// SIMATIC S7-200 project (STEP 7-Micro/WIN), CPU 224 CN REL 02.01

ORGANIZATION_BLOCK MAIN:OB1
TITLE=程序注释
BEGIN
Network 1 // 网络标题
// 网络注释
LD     SM0.1
R      M3.0, 8
R      Q0.0, 10
Network 2
LD     M1.0
R      M1.1, 1
Network 3
LD     M1.1
EU
R      M1.0, 1
R      M3.0, 8
R      Q0.0, 10
Network 4
LD     M1.1
ED
LD     M1.0
EU
OLD
R      M4.5, 2
R      Q0.5, 2
Network 5
LD     M1.1
CALL   SBR_0:SBR0
JMP    15
Network 6
LD     M1.0
EU
A      I0.4
R      M3.0, 8
R      Q0.0, 16
Network 7
LD     M1.0
EU
S      Q0.0, 1
Network 8
LD     M0.0
ED
R      M3.0, 8
R      Q0.0, 16
R      T33, 8
Network 9
LD     M0.0
A      M1.0
AN     M3.4
AN     M3.5
AN     M3.6
AN     M3.7
TON    T37, VW104
Network 10
LD     I0.0
LD     T37
A      M0.0
OLD
R      Q0.0, 1
A      M1.0
AN     Q0.5
AN     M3.5
AN     M3.6
AN     M3.2
A      I0.4
S      Q0.3, 1
R      M3.0, 1
S      M3.1, 1
R      T37, 1
MOVW   +0, T37
Network 11
LD     M3.1
A      I0.3
S      Q0.4, 1
R      Q0.3, 1
Network 12
LD     Q0.4
S      M3.2, 1
Network 13
LD     M3.2
TON    T36, VW102
Network 14
LD     T36
S      Q0.5, 1
R      M3.2, 1
S      M3.5, 1
Network 15
LD     M3.5
A      I0.5
S      Q0.6, 1
S      M3.6, 1
R      M3.5, 1
R      M3.1, 1
R      T36, 1
Network 16
LD     M3.6
TON    T33, VW100
EU
INCD   VD110
Network 17
LD     M0.1
EU
OD>=   VD110, +99999
MOVD   +0, VD110
Network 18
LD     T33
R      Q0.4, 3
R      Q0.5, 1
R      M3.2, 1
R      M3.6, 1
R      M3.1, 1
S      M3.7, 1
S      Q0.0, 1
Network 19
LDN    M1.0
R      Q0.0, 1
Network 20
LDN    M1.0
A      M3.7
R      M3.0, 8
Network 21
LD     M1.0
A      M3.7
R      M3.7, 1
Network 22
LDN    I0.7
A      Q0.0
S      M2.0, 1
Network 23
LD     I0.7
A      M2.0
S      Q0.0, 1
Network 24
LDN    I0.7
R      Q0.0, 1
R      Q0.3, 4
R      M3.5, 3
R      M0.0, 1
Network 25
LD     I0.7
R      M2.0, 1
Network 26
LDN    I0.5
AN     I1.3
R      Q0.4, 3
R      M3.5, 3
Network 27
LBL    15
Network 28
LD     I1.0
=      Q1.0
LD     I1.1
=      Q1.1
END_ORGANIZATION_BLOCK

SUBROUTINE_BLOCK SBR_0:SBR0
TITLE=子程序注释
BEGIN
Network 1 // 网络标题
// 网络注释
LD     M1.1
S      Q0.5, 1
S      M4.5, 1
Network 2
LD     M4.5
A      I0.5
S      Q0.6, 1
END_SUBROUTINE_BLOCK
